// Conversion helper to convert from TcEventSeverity to Intecre.Utilities E_LogSeverity.
FUNCTION INTERNAL F_GetLogSeverityFromTcEventSeverity : E_LogSeverity
VAR_INPUT
  severity : TcEventSeverity;
END_VAR

CASE severity OF

  TcEventSeverity.Verbose   : F_GetLogSeverityFromTcEventSeverity := E_LogSeverity.Debug;
  TcEventSeverity.Info      : F_GetLogSeverityFromTcEventSeverity := E_Logseverity.Info;
  TcEventSeverity.Warning   : F_GetLogSeverityFromTcEventSeverity := E_Logseverity.Warning;
  TcEventSeverity.Error     : F_GetLogSeverityFromTcEventSeverity := E_Logseverity.Error;
  TcEventSeverity.Critical  : F_GetLogSeverityFromTcEventSeverity := E_Logseverity.Error;

END_CASE

END_FUNCTION

(* stored: Version 1.1.0.1, ProductVersion 3.1.4024.12
   POU F_GetLogSeverityFromTcEventSeverity: Id {82b7a67f-d6f1-0024-1b20-fa8788eec8cb}, SpecialFunc None *)
